FUNCTION_BLOCK AUI_UI_TO_UINT (* Composite FB for convert AUI to UINT *)
  (* Standard: 61499-2; Description: Copyright (c) 2026 HR Agrartechnik GmbH This program and the accompanying materials are made available under the terms of the Eclipse Public License 2.0 which is available at https://www.eclipse.org/legal/epl-2.0/ SPDX-License-Identifier: EPL-2.0 *)
  (* Version 1.0, 2026-01-17, Franz Höpfinger, HR Agrartechnik GmbH *)
  PACKAGE adapter::conversion::unidirectional;
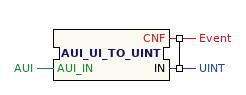
  EVENT_OUTPUT
    CNF WITH IN; (* Confirmation from Adapter *)
  END_EVENT
  VAR_OUTPUT
    IN : UINT; (* Input data from Adapter *)
  END_VAR
  SOCKETS
    AUI_IN : adapter::types::unidirectional::AUI; (* Adapter Input *)
  END_SOCKETS
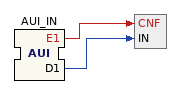
  EVENT_CONNECTIONS
    AUI_IN.E1 TO CNF;
  END_CONNECTIONS
  DATA_CONNECTIONS
    AUI_IN.D1 TO IN;
  END_CONNECTIONS
END_FUNCTION_BLOCK
